TYPE ST_Inverter :
STRUCT
	bDeviceId         : BYTE;
	wStatus	          : E_InverterStatusWord;
	eControl          : E_InverterControlWord;
	errorInv  		  : E_InverterError;           // AVT inverter Error
	sErrorDescription : T_MaxString;
	rSpeed	          : WORD;	
	errorMdb          : MODBUS_ERRORS;  // Modbus Communications error		
END_STRUCT
END_TYPE

(* stored: Version 1.1.0.1, ProductVersion 3.1.4024.12
   DUT ST_Inverter: Id {1bc7dfbe-c465-43ab-9d3e-fb9ebb68c136} *)
